Universal Robots PolyScope program: target_pose_tracking_with_joint_option.urp

Program target_pose_tracking_with_joint_option (createdIn=3.5.4.10845 lastSavedIn=3.5.4.10845 directory=/home/ur/ursim-current/programs installation=default robotSerialNumber=2014359999)
Calibrated DH parameters: a=[-0.000013, -0.610702, -0.570043, 0.000032, 0.000058, 0]; d=[0.128108, 2.4538, -6.32929, 4.038866, 0.115828, 0.092249]; alpha=[1.570687, -0.019005, -0.009774, 1.570693, -1.570802, 0]; deltaTheta=[-0.00004, -0.076204, 0.14266, -0.066295, -0.000042, -0.000021]
BeforeStart
  isJoint := 0
  target_pose := Joint_6_name
  toClose := 0
  toOpen := 0
  Popup Message (haltProgram=false message=Program has started from the beginning :D)
Robot Program (runOnlyOnce=false motionType=MoveJ speed=1.047198 acceleration=1.396263 useActiveTCP=false)
  Script: servoj(get_inverse_kin(target_pose))
  If isJoint≟0
    Script: servoj(get_inverse_kin(target_pose))
  Else 
    Script: servoj(target_pose)
  If toClose≠0
    URCap Gripper (Robotiq_Grippers, Robotiq Inc.) dataModel(position=100.0, force=20.0, speed=100.0, positionInDouble=100.0, forceInDouble=20.0, speedInDouble=100.0, slaveIds=[9], blocking=false); state(isChildrenLocked=true)
  If toOpen≠0
    URCap Gripper (Robotiq_Grippers, Robotiq Inc.) dataModel(position=0.0, force=20.0, speed=100.0, positionInDouble=0.0, forceInDouble=20.0, speedInDouble=100.0, slaveIds=[9], blocking=false); state(isChildrenLocked=true)
  Script: sync()
Thread Thread_1 (runOnlyOnce=false trackProgramExecution=false)
  target_pose := Joint_6_name
  Loop Forever
    tmp := p[0,0,0,0,0,0]
    Script: tmp[0] = read_input_float_register(0)
    Script: tmp[1] = read_input_float_register(1)
    Script: tmp[2] = read_input_float_register(2)
    Script: tmp[3] = read_input_float_register(3)
    Script: tmp[4] = read_input_float_register(4)
    Script: tmp[5] = read_input_float_register(5)
    Script: toClose = read_input_integer_register(1)
    Script: toOpen = read_input_integer_register(2)
    Script: isJoint = read_input_integer_register(3)
    If tmp!=p[0,0,0,0,0,0]
      target_pose := tmp
    Script: sync()
